Fanuc KAREL source: kf00048.KL

-- PROVISIONAL review KL for V940-1; original PC SHA256 2beb661e0f200d0a362e55f08ec0a741fdec15598b1bf151a3178a12b8df7849
-- Incomplete behavior may be omitted. Consult companion uncertainty JSON. Do not deploy.
PROGRAM KF00048
%NOLOCKGROUP
VAR
  I : INTEGER
  J : INTEGER
  X : REAL
  Y : REAL
  B : BOOLEAN
  C : BOOLEAN
  TXT : STRING[80]
  TXT2 : STRING[80]
  STATUS : INTEGER
-- UNRESOLVED_DECL AI type=002010
-- UNRESOLVED_DECL BI type=002010
-- UNRESOLVED_DECL P type=000102
-- UNRESOLVED_DECL JP type=000199
-- UNRESOLVED_DECL PF type=000101
-- UNRESOLVED_DECL V1 type=000013
-- UNRESOLVED_DECL V2 type=000013
BEGIN
  -- UNRESOLVED_PC offsets 5-16; opcodes 2E,23
  -- UNRESOLVED_PC offsets 21-38; opcodes 21,40,41,42
  -- UNRESOLVED_PC offsets 43-70; opcodes 2E,23,7A,40,41,42
  -- UNRESOLVED_PC offsets 75-92; opcodes 2E,23,7A,44
  -- UNRESOLVED_PC offsets 102-106; opcodes 7F
END KF00048
